(* CoDeSys 2.3 export: FSETK14PUMP.EXP *)

(* POU K14/fSetK14Pump, ST *)
FUNCTION fSetK14Pump : BOOL
VAR_INPUT
	State : BOOL;
	PumpID : USINT;
END_VAR
VAR
END_VAR
	MU110DO.K14PumpIsOn[PumpID] := State;
	(*Включить/Выключить реле насоса*)

	PLC160AO.UZSpeed[PumpID]	:= fUZSignalToVoltageOutput(PLC160AI.UZSignal[PumpID]);
	(*Задать управляющее напряжение на насос*)
END_FUNCTION
